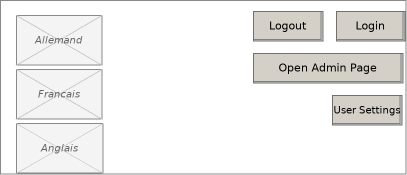
VISUALIZATION Visu2_LanguageUser  // 407x175
    Button (253,53 150x30), "Open Admin Page"
        OnMouseClick: change screen: VisuAdmin
    Button (336,11 69x30), "Login"
        OnMouseClick: VisuUserMgmt Type=Login
    Button (253,11 70x30), "Logout"
        OnMouseClick: VisuUserMgmt Type=Logout
    Button (332,95 70x30), "User Settings"
        OnMouseClick: VisuUserMgmt Type=OpenUserConfiguration
    Image (16,15 86x50), image: Allemand
        OnMouseClick: ChangeLanguage ChangeLanguage=de
    Image (16,69 86x50), image: Francais
        OnMouseClick: ChangeLanguage ChangeLanguage=fr
    Image (16,123 87x50), image: Anglais
        OnMouseClick: ChangeLanguage ChangeLanguage=en
END_VISUALIZATION

(* stored: Version 1.1.0.1, ProductVersion 3.1.4020.12
   Visu Visu2_LanguageUser: Id {a77f1c4c-0c68-4687-88b2-bc14e5e1a3e9} *)
